Fanuc KAREL source: kt00544.KL

-- PROVISIONAL review KL for V940-1; original PC SHA256 f21d35e50f48451f5d9cfadcfdaae7a03b98658baa3091f88dabf372153d7ca8
-- Incomplete behavior may be omitted. Consult companion uncertainty JSON. Do not deploy.
PROGRAM KT00544
%NOLOCKGROUP
-- UNRESOLVED_DECL P1 type=000199
-- UNRESOLVED_DECL P2 type=000106
-- UNRESOLVED_DECL OUT type=000101
BEGIN
  -- V9_ZERO_TABLE_METADATA_HINT layout=0001; no indexed target words; source/name/runtime held
  -- UNRESOLVED_PC offsets 5-20; opcodes 2E,22,32,35
  -- UNRESOLVED_PC offsets 25-59; opcodes 49,7E,49,7E,60,4A
  -- UNRESOLVED_PC offsets 64-68; opcodes 7F
END KT00544
